// TwinCAT 3 PLC project Untitled1
// ProgramVersion: 3.1.4023.0
// libraries:
//   Tc2_Standard, * (Beckhoff Automation GmbH)
//   Tc2_System, * (Beckhoff Automation GmbH)
//   Tc3_Module, * (Beckhoff Automation GmbH)
// project tree:
//   DUTs/ SICK_Process_Data.TcDUT
//   GVLs/ GVL.TcGVL
//   / PlcTask.TcTTO
//   POUs/ MAIN.TcPOU, SICK_Process_Parse.TcPOU
// real-time tasks:
//   TASK PlcTask: cycle T#10ms, priority 20, ADS port 350
//   TASK PlcTask1: cycle T#10ms, priority 21, ADS port 351
// I/O:
//   DEVICE Device 1 (Beckhoff CCAT)
//   DEVICE Device 2 (EtherCAT), AmsNetId 5.104.86.109.3.1
//     Term 1 (EK1200) [EK1200-5000 EtherCAT Power supply (2A E-Bus)]
//       Term 2 (EL6224) [EL6224 (IO Link Master)]
//       Term 3 (EL9011) [EL9011 End Terminal]
// variable links:
//   Untitled1/Untitled1 Instance <-> Device 2 (EtherCAT)/Term 1 (EK1200)/Term 2 (EL6224)
//     PlcTask Inputs/MAIN.bEL6224_Ch1 <-> IO-Link Port1/SubIndex 001

CONFIGURATION Untitled1
    RESOURCE PLC ON TwinCAT3
        TASK PlcTask(INTERVAL := T#10ms, PRIORITY := 21);
        PROGRAM MAIN WITH PlcTask : MAIN;
    END_RESOURCE
END_CONFIGURATION

// ---- DUTs/SICK_Process_Data.TcDUT
TYPE SICK_Process_Data :
STRUCT
	Q	:	BOOL;
	QoR	:	BOOL;
	Emission_Color	:	BYTE;
	value : DINT;
END_STRUCT
END_TYPE

// ---- GVLs/GVL.TcGVL
{attribute 'qualified_only'}
VAR_GLOBAL
	SICK_1_Process: SICK_Process_Data;
END_VAR

// ---- POUs/MAIN.TcPOU
PROGRAM MAIN
VAR
	nSwitchCtrl : BOOL := TRUE;
	nRotateUpper : WORD :=16#8000;
	nRotateLower :WORD :=16#01;
	bEL6224_Ch1 AT%I* : ARRAY[0..1] OF BYTE;
END_VAR

//SICK_Process_Parse(Data:=bEL6224_Ch1 , Process_Data=>GVL.SICK_1_Process );
GVL.SICK_1_Process := SICK_Process_Parse(Data:=bEL6224_Ch1);



























































































































]

END_PROGRAM

// ---- POUs/SICK_Process_Parse.TcPOU
FUNCTION SICK_Process_Parse : SICK_Process_Data
VAR_INPUT
	Data: ARRAY[0..1] OF BYTE;
END_VAR

SICK_Process_Parse.Q := Data[1].0;
SICK_Process_Parse.QoR:= Data[1].2;

SICK_Process_Parse.Emission_Color.0:= Data[1].3;
SICK_Process_Parse.Emission_Color.1:= Data[1].4;
SICK_Process_Parse.Emission_Color.2:= Data[1].5;

SICK_Process_Parse.value.0:= Data[1].6;
SICK_Process_Parse.value.1:= Data[1].7;
SICK_Process_Parse.value.2:= Data[0].0;
SICK_Process_Parse.value.3:= Data[0].1;
SICK_Process_Parse.value.4:= Data[0].2;
SICK_Process_Parse.value.5:= Data[0].3;
SICK_Process_Parse.value.6:= Data[0].4;
SICK_Process_Parse.value.7:= Data[0].5;
SICK_Process_Parse.value.8:= Data[0].6;
SICK_Process_Parse.value.9:= Data[0].7;

RETURN ;

END_FUNCTION
